// LS Electric XG5000 project: Final Python PLC Controll
// PLC LSPLC

PROGRAM NewProgram (task: 스캔 프로그램)

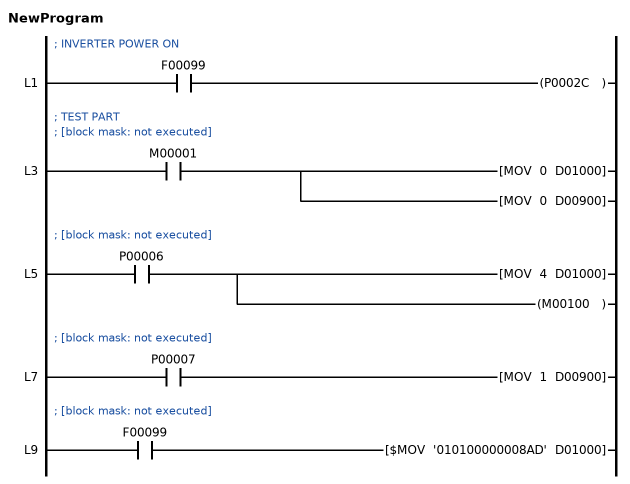
// INVERTER POWER ON
; L1
LOAD      F00099
OUT       P0002C
// TEST PART
; L3 (block mask: not executed)
LOAD      M00001
MOV       0 D01000
MOV       0 D00900
; L5 (block mask: not executed)
LOAD      P00006
MOV       4 D01000
OUT       M00100
; L7 (block mask: not executed)
LOAD      P00007
MOV       1 D00900
; L9 (block mask: not executed)
LOAD      F00099
$MOV      '010100000008AD' D01000